FUNCTION_BLOCK Elevator (* Composite Function Block Type *)
  (* Standard: 61499-2 *)
  (* Version 0.0, 4/20/2019, vshatrov, nxtControl GmbH, template *)
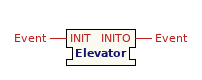
  EVENT_INPUT
    INIT; (* Initialization Request *)
  END_EVENT
  EVENT_OUTPUT
    INITO; (* Initialization Confirm *)
  END_EVENT
  FBS
    model : Model;
    Controller : ControlTS;
    Sensors : Sensors;
  END_FBS
  EVENT_CONNECTIONS
    INIT TO model.INIT;
    INIT TO Controller.INIT;
    model.CNF TO Controller.REQ;
    Controller.CNF TO model.REQ;
    model.INITO TO Sensors.INIT;
    model.UPD TO Sensors.REQ;
    Sensors.CNF TO Controller.UPD;
  END_CONNECTIONS
  DATA_CONNECTIONS
    Controller.MoveUp TO model.motorUp;
    Controller.MoveDown TO model.motorDown;
    model.CarPos TO Sensors.CarPos;
  END_CONNECTIONS
END_FUNCTION_BLOCK
